{attribute 'GeneratedUsingTerminal: EPP1332-0001-0016'}
{attribute addProperty BoxType "EPP1332-0001-0016"}
{attribute addProperty Id "A_0022_EPP1332_0001_0017A_0022_EPP1332_0001_0017_EEFE2EB8378"}
{attribute addProperty CRC "1424085422"}
{attribute addProperty Size "378"}
TYPE A_0021_EPP1332_0001_0016_54E1D1AE EXTENDS EPP1332_1FC0878B :
STRUCT
	{attribute addProperty Name "A_0022(EPP1332-0001-0017)"}
	{attribute addProperty PreviousPort "A_0021(EPP1332-0001-0016) : D"}
	A_0022_EPP1332_0001_0017 : A_0022_EPP1332_0001_0017_EEFE2EB8;
END_STRUCT
END_TYPE

(* stored: Version 1.2.0.0, ProductVersion 3.1.4024.11
   DUT A_0021_EPP1332_0001_0016_54E1D1AE: Id {efe37ae4-c744-485d-bf2e-7e57115da2a2} *)
